KUKA KRL data list: Program1.dat

&ACCESS RV
DEFDAT Program1 PUBLIC

ENDDAT
